Universal Robots PolyScope program: retreat_from_step.urp

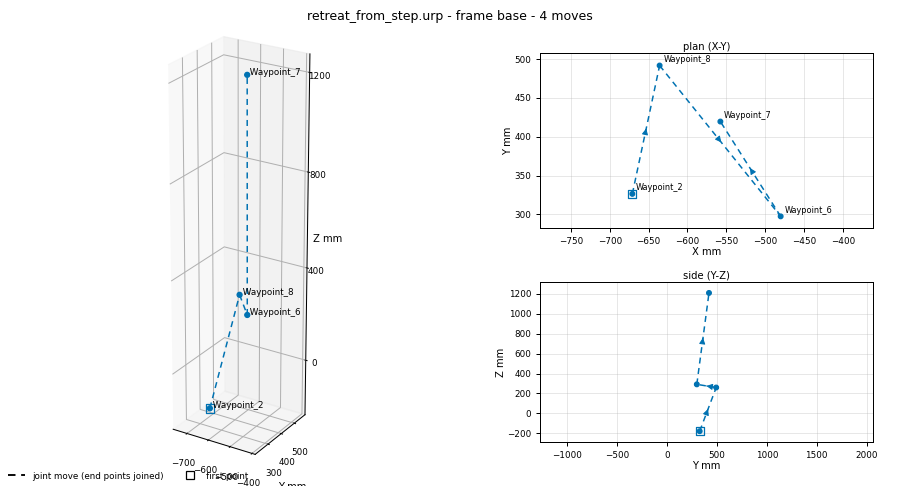
[picture p0: tool path of retreat_from_step.urp in frame base, 4 of 4 moves have a stored position in this frame; points joined in program order, loops and branches not executed]
Program retreat_from_step (installation=default directory=/programs createdIn=5.21.3 lastSavedIn=5.21.3 robotSerialNumber=20246801938)
Calibrated DH parameters: a=[-0.000071, -0.790281, -0.600694, 0.000061, -0.000039, 0]; d=[0.236272, 604.465945, 132.116513, -736.382239, 0.159268, 0.154005]; alpha=[1.570254, -0.000567, 0.000559, 1.571709, -1.56999, 0]; deltaTheta=[0, -0.409357, 7.293326, -0.600784, -0.000001, -0.000001]
InitVariablesNode
Robot Program (runOnlyOnce=false)
  SuppressedNode
    Folder dummy points
      MoveJ speed 60 deg/s, acceleration 80 deg/s^2 (useActiveTCP=true optimoveEnabled=false optiMoveSpeed=0.3 optiMoveAcceleration=0.09) feature=Base
        'right side end points'
        Waypoint Waypoint_1: TCP in base x=-1253.519 y=364.13 z=-67.585 mm, rx=0.018 ry=0.0176 rz=0.7803 rad; joints [-179.095, -181.39, -36.733, -141.231, 46.177, 180.871] deg; TCP offset x=-9.5 y=-328 z=105.73 mm, rx=1.2092 ry=-1.2092 rz=1.2092 rad
        Waypoint Waypoint_3: TCP in base x=-1253.519 y=364.13 z=-129.324 mm, rx=0.018 ry=0.0176 rz=0.7803 rad; joints [-179.093, -185.871, -31.706, -141.776, 46.177, 180.869] deg
      MoveJ speed 60 deg/s, acceleration 80 deg/s^2 (useActiveTCP=true optimoveEnabled=false optiMoveSpeed=0.3 optiMoveAcceleration=0.09) feature=Base
        'left side end points'
        Waypoint Waypoint_4: TCP in base x=-1258.059 y=209.945 z=-65.388 mm, rx=0.0265 ry=-0.0276 rz=2.2505 rad; joints [-170.66, -165.644, -86.102, -104.787, -29.65, 176.354] deg
        Waypoint Waypoint_5: TCP in base x=-1258.059 y=209.945 z=-131.718 mm, rx=0.0265 ry=-0.0276 rz=2.2505 rad; joints [-170.658, -169.867, -82.992, -103.675, -29.649, 176.354] deg
  MoveJ speed 60 deg/s, acceleration 80 deg/s^2 (useActiveTCP=true optimoveEnabled=false optiMoveSpeed=0.3 optiMoveAcceleration=0.09) feature=Base
    Waypoint Waypoint_2: TCP in base x=-670.966 y=326.422 z=-178.215 mm, rx=0.0098 ry=0.0257 rz=1.6447 rad; joints [-167.814, -172.971, -116.48, -67.413, 7.981, 178.204] deg
  MoveJ speed 60 deg/s, acceleration 80 deg/s^2 (useActiveTCP=true optimoveEnabled=false optiMoveSpeed=0.3 optiMoveAcceleration=0.09) feature=Base
    Waypoint Waypoint_8: TCP in base x=-635.85 y=491.712 z=259.684 mm, rx=-0.4995 ry=-0.7883 rz=1.854 rad; joints [-203.235, -128.315, -150.467, -80.055, -46.632, 133.613] deg
    Waypoint Waypoint_6: TCP in base x=-479.957 y=297.468 z=291.375 mm, rx=-0.7812 ry=-1.774 rz=1.7129 rad; joints [-222.662, -82.07, -155.488, -122.893, -85.563, 87.81] deg
  MoveJ speed 60 deg/s, acceleration 80 deg/s^2 (useActiveTCP=true optimoveEnabled=false optiMoveSpeed=0.3 optiMoveAcceleration=0.09) feature=Base
    Waypoint Waypoint_7: TCP in base x=-557.589 y=419.56 z=1207.727 mm, rx=-0.5026 ry=-0.0558 rz=1.8139 rad; joints [-165.719, -50.766, -121.227, -102.266, 18.039, 76.633] deg
  SafeHome (positionOptionType=SPEED_AND_ACCELERATION speed=1.047198 acceleration=1.396263 nextMotionTime=2)
